// TwinCAT 3 PLC project BE_RobertWeinhandl
// ProgramVersion: 3.1.4023.0
// libraries:
//   EfficientIO Communicator, * (EfficientIO)
//   Lynus Energy Basic, * (Lynus AG)
//   Lynus Energy ModbusTCP, * (Lynus AG)
//   Lynus Standards, * (Lynus AG)
//   Tc2_MBus, * (Beckhoff Automation GmbH)
//   Tc2_Standard, * (Beckhoff Automation GmbH)
//   Tc2_System, * (Beckhoff Automation GmbH)
//   Tc2_SystemCX, * (Beckhoff Automation GmbH)
//   Tc2_Utilities, * (Beckhoff Automation GmbH)
//   Tc3_IotBase, * (Beckhoff Automation GmbH)
//   Tc3_JsonXml, * (Beckhoff Automation GmbH)
//   Tc3_Module, * (Beckhoff Automation GmbH)
// project tree:
//   / FastTask.TcTTO, MiddleTask.TcTTO, SlowTask.TcTTO
//   FB/ FB_FroniusSymo_JSON.TcPOU, FB_FroniusSymo_JSON_Helper.TcPOU, FB_KL6781_MBus_Master.TcPOU, FB_Shelly_3EM.TcPOU, FB_Shelly_3EM_Helper.TcPOU, FB_Shelly_Pro4PM.TcPOU, FB_Shelly_Pro4PM_Helper.TcPOU
//   POUs/ Logic.TcPOU (excluded from build), prgComEffIO.TcPOU, prgGrid.TcPOU, prgMain.TcPOU, prgPV.TcPOU, prgRWEffIO.TcPOU (not stored), prgShelly.TcPOU, prgSmartMeter.TcPOU (excluded from build), prgVarEffIO.TcPOU (not stored)
// real-time tasks:
//   TASK MiddleTask: cycle T#10ms, priority 8, ADS port 350
//   TASK FastTask: cycle T#5ms, priority 6, ADS port 351
//   TASK SlowTask: cycle T#20ms, priority 10, ADS port 352
// I/O:
//   DEVICE Device 1 (Beckhoff CCAT)
//   DEVICE Device 2 (CX-BK)
//     Box 1 (CX-BK)

CONFIGURATION BE_RobertWeinhandl
    RESOURCE PLC ON TwinCAT3
        TASK FastTask(INTERVAL := T#5ms, PRIORITY := 6);
        TASK MiddleTask(INTERVAL := T#10ms, PRIORITY := 8);
        TASK SlowTask(INTERVAL := T#20ms, PRIORITY := 10);
        PROGRAM prgRWEffIO WITH FastTask : prgRWEffIO;
        PROGRAM prgVarEffIO WITH FastTask : prgVarEffIO;
        PROGRAM prgShelly WITH MiddleTask : prgShelly;
        PROGRAM prgPV WITH MiddleTask : prgPV;
        PROGRAM prgGrid WITH MiddleTask : prgGrid;
        PROGRAM prgMain WITH MiddleTask : prgMain;
        PROGRAM prgComEffIO WITH SlowTask : prgComEffIO;
    END_RESOURCE
END_CONFIGURATION

// ---- POUs/prgShelly.TcPOU
PROGRAM prgShelly
VAR
	// Charging Cabel 3-phase, 400V
	fbCS						: FB_Shelly_3EM;
	
	lrPowerCSTotal				: LREAL;	//{#lynus.ag#()}
	lrPowerCSTotalkW			: LREAL;	//{#lynus.ag#()}
	lrEnergyCSTotal				: LREAL;	//{#lynus.ag#()}
	lrPowerCSL1					: LREAL;	//{#lynus.ag#()}
	lrPowerCSL2					: LREAL;	//{#lynus.ag#()}
	lrPowerCSL3					: LREAL;	//{#lynus.ag#()}
	lrCurrentCSL1				: LREAL;	//{#lynus.ag#()}
	lrCurrentCSL2				: LREAL;	//{#lynus.ag#()}
	lrCurrentCSL3				: LREAL;	//{#lynus.ag#()}
	lrVoltageCSL1				: LREAL;	//{#lynus.ag#()}
	lrVoltageCSL2				: LREAL;	//{#lynus.ag#()}
	lrVoltageCSL3				: LREAL;	//{#lynus.ag#()}
	lrEnergyCSL1				: LREAL;	//{#lynus.ag#()}
	lrEnergyCSL2				: LREAL;	//{#lynus.ag#()}
	lrEnergyCSL3				: LREAL;	//{#lynus.ag#()}
	
	// Garage and Pool
	fbGarage					: FB_Shelly_3EM;
	
	lrPowerGarageTotal			: LREAL;	//{#lynus.ag#()}
	lrPowerGarageTotalkW		: LREAL;	//{#lynus.ag#()}
	lrEnergyGarageTotal			: LREAL;	//{#lynus.ag#()}
	lrPowerGarageL1				: LREAL;	//{#lynus.ag#()}
	lrPowerGarageL2				: LREAL;	//{#lynus.ag#()}
	lrPowerGarageL3				: LREAL;	//{#lynus.ag#()}
	lrCurrentGarageL1			: LREAL;	//{#lynus.ag#()}
	lrCurrentGarageL2			: LREAL;	//{#lynus.ag#()}
	lrCurrentGarageL3			: LREAL;	//{#lynus.ag#()}
	lrVoltageGarageL1			: LREAL;	//{#lynus.ag#()}
	lrVoltageGarageL2			: LREAL;	//{#lynus.ag#()}
	lrVoltageGarageL3			: LREAL;	//{#lynus.ag#()}
	lrEnergyGarageL1			: LREAL;	//{#lynus.ag#()}
	lrEnergyGarageL2			: LREAL;	//{#lynus.ag#()}
	lrEnergyGarageL3			: LREAL;	//{#lynus.ag#()}
		
	// UV Keller
	fbUVKeller						: FB_Shelly_3EM;
	fbUVKellerCounter				: FB_EnergyCounter;
	
	lrPowerUVKellerTotal			: LREAL;	//{#lynus.ag#()}
	lrPowerUVKellerTotalkW			: LREAL;	//{#lynus.ag#()}
	lrEnergyUVKellerTotal			: LREAL;	//{#lynus.ag#()}
	lrPowerUVKellerL1				: LREAL;	//{#lynus.ag#()}
	lrPowerUVKellerL2				: LREAL;	//{#lynus.ag#()}
	lrPowerUVKellerL3				: LREAL;	//{#lynus.ag#()}
	lrCurrentUVKellerL1			: LREAL;	//{#lynus.ag#()}
	lrCurrentUVKellerL2			: LREAL;	//{#lynus.ag#()}
	lrCurrentUVKellerL3			: LREAL;	//{#lynus.ag#()}
	lrVoltageUVKellerL1			: LREAL;	//{#lynus.ag#()}
	lrVoltageUVKellerL2			: LREAL;	//{#lynus.ag#()}
	lrVoltageUVKellerL3			: LREAL;	//{#lynus.ag#()}
	lrEnergyUVKellerL1				: LREAL;	//{#lynus.ag#()}
	lrEnergyUVKellerL2				: LREAL;	//{#lynus.ag#()}
	lrEnergyUVKellerL3				: LREAL;	//{#lynus.ag#()}
END_VAR

VAR PERSISTENT
// trigger command execution
	bEnableCS 				: BOOL;		//{#lynus.ag#()}
	bEnableGarage			: BOOL;		//{#lynus.ag#()}
	bEnableUVKeller			: BOOL;		//{#lynus.ag#()}
	lrCounterUVKeller		: LREAL;	//{#lynus.ag#()}
END_VAR

// Charging Cable 3-phase, 400V
fbCS(
	bStart:= bEnableCS, 
	tDelayRequest:= T#20S, 
	sHostname:= '192.168.0.31', 
	bValidResult=> , 
	bBusy=> , 
	bError=> , 
	bDone=> , 
	hrErrorCode=> ,
	lrtotalpower=> lrPowerCSTotal,
	lrpowerL1=> lrPowerCSL1,
	lrpowerL2=> lrPowerCSL2,
	lrpowerL3=> lrPowerCSL3,
	lrcurrentL1=> lrCurrentCSL1,
	lrcurrentL2=> lrCurrentCSL2,
	lrcurrentL3=> lrCurrentCSL3,
	lrvoltageL1=> lrVoltageCSL1,
	lrvoltageL2=> lrVoltageCSL2,
	lrvoltageL3=> lrVoltageCSL3,
	lrenergyL1=> lrEnergyCSL1,
	lrenergyL2=> lrEnergyCSL2,
	lrenergyL3=> lrEnergyCSL3 );

	// re-calc to kW
	lrPowerCSTotalkW := lrPowerCSTotal / 1000;
	// sum-up energy
	lrEnergyCSTotal :=  lrEnergyCSL1 + lrEnergyCSL2 + lrEnergyCSL3;


// Garage and Pool
fbGarage(
	bStart:= bEnableGarage, 
	tDelayRequest:= T#20S, 
	sHostname:= '192.168.0.30', 
	bValidResult=> , 
	bBusy=> , 
	bError=> , 
	bDone=> , 
	hrErrorCode=> ,
	lrtotalpower=> lrPowerGarageTotal,
	lrpowerL1=> lrPowerGarageL1,
	lrpowerL2=> lrPowerGarageL2,
	lrpowerL3=> lrPowerGarageL3,
	lrcurrentL1=> lrCurrentGarageL1,
	lrcurrentL2=> lrCurrentGarageL2,
	lrcurrentL3=> lrCurrentGarageL3,
	lrvoltageL1=> lrVoltageGarageL1,
	lrvoltageL2=> lrVoltageGarageL2,
	lrvoltageL3=> lrVoltageGarageL3,
	lrenergyL1=> lrEnergyGarageL1,
	lrenergyL2=> lrEnergyGarageL2,
	lrenergyL3=> lrEnergyGarageL3 );

	// re-calc to kW
	lrPowerGarageTotalkW := lrPowerGarageTotal / 1000;
	// sum-up energy
	lrEnergyGarageTotal :=  lrEnergyGarageL1 + lrEnergyGarageL2 + lrEnergyGarageL3;

	
// UVKeller
fbUVKeller(
	bStart:= bEnableUVKeller, 
	tDelayRequest:= T#20S, 
	sHostname:= '192.168.0.35', 
	bValidResult=> , 
	bBusy=> , 
	bError=> , 
	bDone=> , 
	hrErrorCode=> ,
	lrtotalpower=> ,
	lrpowerL1=> ,
	lrpowerL2=> ,
	lrpowerL3=> ,
	lrcurrentL1=> lrCurrentUVKellerL1,
	lrcurrentL2=> lrCurrentUVKellerL2,
	lrcurrentL3=> lrCurrentUVKellerL3,
	lrvoltageL1=> lrVoltageUVKellerL1,
	lrvoltageL2=> lrVoltageUVKellerL2,
	lrvoltageL3=> lrVoltageUVKellerL3,
	lrenergyL1=> lrEnergyUVKellerL1,
	lrenergyL2=> lrEnergyUVKellerL2,
	lrenergyL3=> lrEnergyUVKellerL3 );
	
lrPowerUVKellerTotal := fbUVKeller.lrtotalpower * (-1);

	// re-calc to kW
	lrPowerUVKellerTotalkW := lrPowerUVKellerTotal / 1000;

// EnergyCounter UV Keller
fbUVKellerCounter(
	byActiveTariff:= 1, 
	lrPowerInput:= lrPowerUVKellerTotalkW, 
	lrTotalCounterEnergy_Consumption=> , 
	lrTotalCounterEnergy_Production=> , 
	lrCounterEnergyT1_Consumption=> , 
	lrCounterEnergyT2_Consumption=> , 
	lrCounterEnergyT1_Production=> , 
	lrCounterEnergyT2_Production=> );
	
IF fbUVKellerCounter.lrTotalCounterEnergy_Consumption > lrCounterUVKeller THEN  	
	lrCounterUVKeller := fbUVKellerCounter.lrTotalCounterEnergy_Consumption;
END_IF

END_PROGRAM

// ---- FB/FB_Shelly_3EM.TcPOU
FUNCTION_BLOCK FB_Shelly_3EM
VAR_INPUT
	bStart				: BOOL;
	tDelayRequest		: TIME;		//Timer for delay before start with the next read or write Request
	sHostname			: STRING(255);		//Hostname or IP Adress from the Server
END_VAR

VAR_IN_OUT
END_VAR

VAR_OUTPUT
	bValidResult		: BOOL;							//Valid Result received from Server
    bBusy				: BOOL;							//Function is Busy
    bError				: BOOL;							//Error sucess
	bDone				: BOOL;							//True after the decoding from the received Json File
	bConnected			: BOOL;							//Connection to the Server
	lrtotalpower		: LREAL;						//Received Value
	lrpowerL1			: LREAL;
	lrcurrentL1			: LREAL;
	lrvoltageL1			: LREAL;
	lrenergyL1			: LREAL;
	lrpowerL2			: LREAL;
	lrcurrentL2			: LREAL;
	lrvoltageL2			: LREAL;
	lrenergyL2			: LREAL;
	lrpowerL3			: LREAL;
	lrcurrentL3			: LREAL;
	lrvoltageL3			: LREAL;
	lrenergyL3			: LREAL;
	hrErrorCode       	: HRESULT;						//Error Result from Http Client
END_VAR

VAR
	fbClient			: FB_IotHttpClient;
	fbHttpGet			: FB_Shelly_3EM_Helper;
	timStartRequest		: TON;							//Timer to Start the Request
	FPStartRequest		: R_TRIG;						//Internal positive Edge
	FPDone				: R_TRIG;						//Internal positive Edge
	FNStart				: F_TRIG;						//Internal negative Edge
END_VAR

(*------------------------------------------------------------------------------------Configure HTTP Client------------------------------------------------------------------------------------------------------*)

fbClient.sHostName := sHostname;
fbClient.tConnectionTimeout := T#30S;

IF NOT fbClient.bConfigured THEN 
	fbClient.nHostPort:= 80;
	fbClient.bKeepAlive := TRUE;
	fbClient.tConnectionTimeout := T#30S;
END_IF


//Timer to start the Request
FPStartRequest(CLK:= bStart, Q=> );
	timStartRequest(IN:= fbClient.bConfigured AND bStart AND NOT timStartRequest.Q, PT:= tDelayRequest, Q=> , ET=> );
		IF ((timStartRequest.Q AND NOT bBusy) OR (FPStartRequest.Q AND NOT bBusy AND fbClient.bConfigured)) THEN fbHttpGet.bSend := TRUE; END_IF

				
//Http Get Function
fbHttpGet(
	lrtotalpower => lrtotalpower, 
	lrpowerL1 => lrpowerL1,
	lrcurrentL1 => lrcurrentL1,
	lrvoltageL1 => lrvoltageL1,
	lrenergyL1 => lrenergyL1,
	lrpowerL2 => lrpowerL2,
	lrcurrentL2 => lrcurrentL2,
	lrvoltageL2 => lrvoltageL2,
	lrenergyL2 => lrenergyL2,
	lrpowerL3 => lrpowerL3,
	lrcurrentL3 => lrcurrentL3,
	lrvoltageL3 => lrvoltageL3,
	lrenergyL3 => lrenergyL3,
	bSend:= , 
	fbClient:= fbClient, 
	bBusy=> bBusy, 
	bError=> ,
	sContentStatus=> ,
	sContentM0=> ,
	sContentM1=> ,
	sContentM2=> );


fbHttpGet.bSend := FALSE;

FPDone(CLK:= bDone, Q=> );

(*
//Http Client
FNStart(CLK:= bStart, Q=> );
	IF FNStart.Q THEN fbClient.Disconnect(); END_IF
*)

fbClient.Execute();

//Error
IF fbHttpGet.bError OR fbClient.bError THEN bError := TRUE; ELSE bError := FALSE; END_IF	
	hrErrorCode := fbClient.hrErrorCode;

END_FUNCTION_BLOCK

// ---- FB/FB_Shelly_3EM_Helper.TcPOU
FUNCTION_BLOCK FB_Shelly_3EM_Helper
VAR_INPUT
	bSend				: BOOL;
END_VAR

VAR_IN_OUT
	fbClient			: FB_IotHttpClient;
END_VAR

VAR_OUTPUT
	bBusy				: BOOL;
	bError				: BOOL;
	lrtotalpower		: LREAL;
	lrpowerL1			: LREAL;
	lrcurrentL1			: LREAL;
	lrvoltageL1			: LREAL;
	lrenergyL1			: LREAL;
	lrpowerL2			: LREAL;
	lrcurrentL2			: LREAL;
	lrvoltageL2			: LREAL;
	lrenergyL2			: LREAL;
	lrpowerL3			: LREAL;
	lrcurrentL3			: LREAL;
	lrvoltageL3			: LREAL;
	lrenergyL3			: LREAL;
END_VAR

VAR
	fbRequestStatus		: FB_IotHttpRequest;
	fbRequestMeter0		: FB_IotHttpRequest;
	fbRequestMeter1		: FB_IotHttpRequest;
	fbRequestMeter2		: FB_IotHttpRequest;
	fbJson				: FB_JsonDomParser;
	nState				: UDINT;
	RisingEdge			: R_TRIG;
	timTimeout			: TON;
	tTimeOut			: TIME := T#50S;
	bGetContentResult	: BOOL;
	sContentStatus		: STRING(511);
	sContentM0			: STRING(511);
	sContentM1			: STRING(511);
	sContentM2			: STRING(511);
	
	bGetJsonResult		: BOOL;
	jsonDoc				: SJsonValue;
	jsonVal				: SJsonValue;
	
	nReqCount			: UDINT;	
	nResCount			: UDINT;
	nValidResCount		: UDINT;
	nErrCount			: UDINT;
END_VAR

//Timer for Timeout
timTimeout(IN:= nState = 1 AND bBusy, PT:= tTimeOut, Q=> , ET=> );
	IF timTimeout.Q THEN 
		nState := 0;
		bBusy := FALSE;
	END_IF

RisingEdge(CLK:= bSend );
CASE nState OF
0:	
	IF RisingEdge.Q THEN 
		IF 
			fbRequestStatus.SendRequest(sUri:='/status', fbClient:=fbClient, eRequestType:=ETcIotHttpRequestType.HTTP_Get, 0, 0, 0) AND
			fbRequestMeter0.SendRequest(sUri:='/emeter/0', fbClient:=fbClient, eRequestType:=ETcIotHttpRequestType.HTTP_Get, 0, 0, 0) AND 
			fbRequestMeter1.SendRequest(sUri:='/emeter/1', fbClient:=fbClient, eRequestType:=ETcIotHttpRequestType.HTTP_Get, 0, 0, 0) AND
			fbRequestMeter2.SendRequest(sUri:='/emeter/2', fbClient:=fbClient, eRequestType:=ETcIotHttpRequestType.HTTP_Get, 0, 0, 0) THEN				
			nState:= 1;
			nReqCount:= nReqCount+1;
			bBusy:= TRUE;
			bError:= FALSE;
		END_IF					
	END_IF
1:
	IF NOT fbRequestMeter0.bBusy AND NOT fbRequestMeter1.bBusy AND NOT fbRequestMeter2.bBusy AND NOT fbRequestStatus.bBusy THEN
		bError:= TRUE;
		IF NOT fbRequestMeter0.bError THEN				 
			bGetContentResult:= fbRequestMeter0.GetContent(pContent:= ADR(sContentM0), nContentSize:= SIZEOF(sContentM0), bSetNullTermination:= TRUE);
			IF fbRequestMeter0.nStatusCode >= 200 AND fbRequestMeter0.nStatusCode < 300 THEN
				bGetJsonResult:= FALSE;
				jsonDoc:= fbRequestMeter0.GetJsonDomContent(fbJson);
				IF jsonDoc <> 0 THEN
					bGetJsonResult:= TRUE;
					IF fbJson.HasMember(jsonDoc, 'power')  THEN
						jsonVal:= fbJson.FindMember(jsonDoc, 'power');
						nValidResCount:= nValidResCount+1;
						IF fbJson.IsDouble(jsonVal) THEN							
							lrpowerL1:= fbJson.GetDouble(jsonVal);									
						END_IF
						jsonVal:= fbJson.FindMember(jsonDoc, 'current');
						nValidResCount:= nValidResCount+1;
						IF fbJson.IsDouble(jsonVal) THEN							
							lrcurrentL1:= fbJson.GetDouble(jsonVal);									
						END_IF
						jsonVal:= fbJson.FindMember(jsonDoc, 'voltage');
						nValidResCount:= nValidResCount+1;
						IF fbJson.IsDouble(jsonVal) THEN							
							lrvoltageL1:= fbJson.GetDouble(jsonVal);									
						END_IF
						jsonVal:= fbJson.FindMember(jsonDoc, 'total');
						nValidResCount:= nValidResCount+1;
						IF fbJson.IsDouble(jsonVal) THEN							
							lrenergyL1:= fbJson.GetDouble(jsonVal);									
						END_IF	
						bError:= FALSE;
						END_IF
					END_IF						
				nResCount:= nResCount+1;			
				END_IF
		END_IF
		
		IF NOT fbRequestMeter1.bError THEN				 
			bGetContentResult:= fbRequestMeter1.GetContent(pContent:= ADR(sContentM1), nContentSize:= SIZEOF(sContentM1), bSetNullTermination:= TRUE);
			IF fbRequestMeter1.nStatusCode >= 200 AND fbRequestMeter1.nStatusCode < 300 THEN
				bGetJsonResult:= FALSE;
				jsonDoc:= fbRequestMeter1.GetJsonDomContent(fbJson);
				IF jsonDoc <> 0 THEN
					bGetJsonResult:= TRUE;
					IF fbJson.HasMember(jsonDoc, 'power')  THEN
						jsonVal:= fbJson.FindMember(jsonDoc, 'power');
						nValidResCount:= nValidResCount+1;
						IF fbJson.IsDouble(jsonVal) THEN							
							lrpowerL2:= fbJson.GetDouble(jsonVal);									
						END_IF
						jsonVal:= fbJson.FindMember(jsonDoc, 'current');
						nValidResCount:= nValidResCount+1;
						IF fbJson.IsDouble(jsonVal) THEN							
							lrcurrentL2:= fbJson.GetDouble(jsonVal);									
						END_IF
						jsonVal:= fbJson.FindMember(jsonDoc, 'voltage');
						nValidResCount:= nValidResCount+1;
						IF fbJson.IsDouble(jsonVal) THEN							
							lrvoltageL2:= fbJson.GetDouble(jsonVal);									
						END_IF
						jsonVal:= fbJson.FindMember(jsonDoc, 'total');
						nValidResCount:= nValidResCount+1;
						IF fbJson.IsDouble(jsonVal) THEN							
							lrenergyL2:= fbJson.GetDouble(jsonVal);									
						END_IF	
						bError:= FALSE;
						END_IF
					END_IF						
				nResCount:= nResCount+1;			
				END_IF
		END_IF
		
		IF NOT fbRequestMeter2.bError THEN				 
			bGetContentResult:= fbRequestMeter2.GetContent(pContent:= ADR(sContentM2), nContentSize:= SIZEOF(sContentM2), bSetNullTermination:= TRUE);
			IF fbRequestMeter2.nStatusCode >= 200 AND fbRequestMeter2.nStatusCode < 300 THEN
				bGetJsonResult:= FALSE;
				jsonDoc:= fbRequestMeter2.GetJsonDomContent(fbJson);
				IF jsonDoc <> 0 THEN
					bGetJsonResult:= TRUE;
					IF fbJson.HasMember(jsonDoc, 'power')  THEN
						jsonVal:= fbJson.FindMember(jsonDoc, 'power');
						nValidResCount:= nValidResCount+1;
						IF fbJson.IsDouble(jsonVal) THEN							
							lrpowerL3:= fbJson.GetDouble(jsonVal);									
						END_IF
						jsonVal:= fbJson.FindMember(jsonDoc, 'current');
						nValidResCount:= nValidResCount+1;
						IF fbJson.IsDouble(jsonVal) THEN							
							lrcurrentL3:= fbJson.GetDouble(jsonVal);									
						END_IF
						jsonVal:= fbJson.FindMember(jsonDoc, 'voltage');
						nValidResCount:= nValidResCount+1;
						IF fbJson.IsDouble(jsonVal) THEN							
							lrvoltageL3:= fbJson.GetDouble(jsonVal);									
						END_IF
						jsonVal:= fbJson.FindMember(jsonDoc, 'total');
						nValidResCount:= nValidResCount+1;
						IF fbJson.IsDouble(jsonVal) THEN							
							lrenergyL3:= fbJson.GetDouble(jsonVal);									
						END_IF	
						bError:= FALSE;
						END_IF
					END_IF						
				nResCount:= nResCount+1;			
				END_IF
		END_IF
		
		IF NOT fbRequestStatus.bError THEN				 
			bGetContentResult:= fbRequestStatus.GetContent(pContent:= ADR(sContentStatus), nContentSize:= SIZEOF(sContentStatus), bSetNullTermination:= TRUE);
			IF fbRequestStatus.nStatusCode >= 200 AND fbRequestStatus.nStatusCode < 300 THEN
				bGetJsonResult:= FALSE;
				jsonDoc:= fbRequestStatus.GetJsonDomContent(fbJson);
				IF jsonDoc <> 0 THEN
					bGetJsonResult:= TRUE;
					IF fbJson.HasMember(jsonDoc, 'total_power')  THEN
						jsonVal:= fbJson.FindMember(jsonDoc, 'total_power');
						nValidResCount:= nValidResCount+1;
						IF fbJson.IsDouble(jsonVal) THEN							
							lrtotalpower:= fbJson.GetDouble(jsonVal);									
						END_IF
						bError:= FALSE;
					END_IF
				END_IF		
				nResCount:= nResCount+1;			
			END_IF
		END_IF
		
		nState:= 0;
		bBusy:= FALSE;
		IF bError THEN
			nErrCount:= nErrCount+1;
		END_IF
	END_IF  	
END_CASE

END_FUNCTION_BLOCK

// ---- POUs/prgPV.TcPOU
PROGRAM prgPV
VAR
	fbPV					: FB_Symo_PV_Inverter_FLOAT_1_DM_1_Inverter;
	fbPVInt					: FB_PV_Power;
	fbPVCounter				: FB_EnergyCounter;
	lrPowerPV				: LREAL;				//{#lynus.ag#()}
	byErrorWarningPV		: BYTE;					//{#lynus.ag#()}
	bReadyPD_PV				: BOOL;					//{#lynus.ag#()}
	byErrorWarningPD_PV		: BYTE;					//{#lynus.ag#()}
	rHeartbeat_PD_PV		: REAL;					//{#lynus.ag#()}
END_VAR

VAR PERSISTENT
	lrCounterPV				: LREAL;				//{#lynus.ag#()}
END_VAR

fbPV(
	bEnable:= TRUE, 
	sIPAdress:= '192.168.0.102', 
	byUnitID_Inverter:= 1, 
	stDataSymo10=> , 
	stDataEMPower_PV=> , 
	stDataEMCounter_PV=> , 
	diNrOfEM_OUT_PV=> );

fbPVInt(
	bEnable:= TRUE, 
	bPowerDataInvers:= , 
	diNrOfEM_IN_PV:= fbPV.diNrOfEM_OUT_PV, 
	stDataPv=> , 
	diNrOfPv_OUT=> );
	
lrPowerPV := fbPVInt.stDataPv.lrPower;
	byErrorWarningPV := fbPVInt.stDataPv.byErrorWarning;

// EnergyCounter
fbPVCounter(
	byActiveTariff:= 1, 
	lrPowerInput:= 0 - lrPowerPV, 
	lrTotalCounterEnergy_Consumption=> , 
	lrTotalCounterEnergy_Production=> , 
	lrCounterEnergyT1_Consumption=> , 
	lrCounterEnergyT2_Consumption=> , 
	lrCounterEnergyT1_Production=> , 
	lrCounterEnergyT2_Production=> );
	
IF fbPVCounter.lrTotalCounterEnergy_Production > lrCounterPV THEN  	
	lrCounterPV := fbPVCounter.lrTotalCounterEnergy_Production;
END_IF

END_PROGRAM

// ---- POUs/prgGrid.TcPOU
PROGRAM prgGrid
VAR
	lrPowerGridkW		: LREAL;	//{#lynus.ag#()}
END_VAR

lrPowerGridkW := prgShelly.lrPowerCSTotalkW + prgShelly.lrPowerGarageTotalkW + prgShelly.lrPowerUVKellerTotalkW - prgPV.lrPowerPV;

END_PROGRAM

// ---- POUs/prgMain.TcPOU
PROGRAM prgMain
VAR
	fb_Reboot		: NT_reboot;
	m_Reboot		: BOOL:=FALSE;
END_VAR

fb_Reboot(	netid := '',
			delay := 2,
			start := m_Reboot);

END_PROGRAM

// ---- POUs/prgComEffIO.TcPOU
PROGRAM prgComEffIO
VAR
	fbCom		: FB_MqttCommunicator_V2;
END_VAR

fbCom(
	bConnect:= TRUE, 
	strAuthKey := 'BE736352867778',
	sUserName:= '9e35a788-9544-4d1e-a992-8e2eed9a2bf4', 
	sUserPassword:= 'b22fd0d3-05b2-481b-ab97-9bb6cc09e5f2', 
	eSavePositionCertificate:= eSavePositionOnPLC.ePostionHardDisk, 
	bConnected=> , 
	bError=> , 
	hrErrorCode=> , 
	eConnectionState=> , 
	eErrorMessage_Out=> );

END_PROGRAM

// ---- FB/FB_FroniusSymo_JSON.TcPOU
FUNCTION_BLOCK FB_FroniusSymo_JSON
VAR_INPUT
	bStart				: BOOL;
	tDelayRequest		: TIME := T#3S;	//Timer for delay before start with the next read or write Request
	sHostname			: STRING(255);		//Hostname or IP Adress from the Server
END_VAR

VAR_IN_OUT
END_VAR

VAR_OUTPUT
	bValidResult				: BOOL;															//Valid Result received from Server
    bBusy						: BOOL;															//Function is Busy
    bError						: BOOL;															//Error sucess
	bDone						: BOOL;															//True after the decoding from the received Json File
	bConnected					: BOOL;															//Connection to the Server
	lrpowerP1					: LREAL;														//Received Value
	lrvoltageP1					: LREAL;														//Received Value
	lrenergyP1					: LREAL;														//Received Value
	lrpowerP2					: LREAL;														//Received Value
	lrvoltageP2					: LREAL;														//Received Value
	lrenergyP2					: LREAL;
	lrpowerP3					: LREAL;														//Received Value
	lrvoltageP3					: LREAL;														//Received Value
	lrenergyP3					: LREAL;
	lrpowerP4					: LREAL;														//Received Value
	lrvoltageP4					: LREAL;														//Received Value
	lrenergyP4					: LREAL;	
	hrErrorCode       			: HRESULT;														//Error Result from Http Client
END_VAR

VAR
	fbClient					: FB_IotHttpClient;
	fbHttpGet					: FB_FroniusSymo_JSON_Helper;
	timStartRequest				: TON;															//Timer to Start the Request
	FPStartRequest				: R_TRIG;														//Internal positive Edge
	FPDone						: R_TRIG;														//Internal positive Edge
	FNStart						: F_TRIG;														//Internal negative Edge
END_VAR

(*------------------------------------------------------------------------------------Configure HTTP Client------------------------------------------------------------------------------------------------------*)

fbClient.sHostName := sHostname;
fbClient.tConnectionTimeout := tDelayRequest;

IF NOT fbClient.bConfigured THEN 
	fbClient.nHostPort:= 80;
	fbClient.bKeepAlive := TRUE;
	fbClient.tConnectionTimeout := T#2S;
END_IF


//Timer to start the Request
FPStartRequest(CLK:= bStart, Q=> );
	timStartRequest(IN:= fbClient.bConfigured AND bStart AND NOT timStartRequest.Q, PT:= tDelayRequest, Q=> , ET=> );
		IF ((timStartRequest.Q AND NOT bBusy) OR (FPStartRequest.Q AND NOT bBusy AND fbClient.bConfigured)) THEN fbHttpGet.bSend := TRUE; END_IF

				
//Http Get Function
fbHttpGet(
	lrapowerP1 => lrpowerP1, 
	lrvoltageP1 => lrvoltageP1, 
	lraenergyP1 => lrenergyP1,
	lrapowerP2 => lrpowerP2, 
	lrvoltageP2 => lrvoltageP2, 
	lraenergyP2 => lrenergyP2,
	lrapowerP3 => lrpowerP3, 
	lrvoltageP3 => lrvoltageP3, 
	lraenergyP3 => lrenergyP3,
	lrapowerP4 => lrpowerP4, 
	lrvoltageP4 => lrvoltageP4, 
	lraenergyP4 => lrenergyP4, 
	bSend:= , 
	fbClient:= fbClient, 
	bBusy=> bBusy, 
	bError=> ,
	sContentS0=> ,
	sContentS1=> ,
	sContentS2=> ,
	sContentS3=> );


fbHttpGet.bSend := FALSE;

FPDone(CLK:= bDone, Q=> );

//Http Client
FNStart(CLK:= bStart, Q=> );
	IF FNStart.Q THEN fbClient.Disconnect(); END_IF

fbClient.Execute();

//Error
IF fbHttpGet.bError OR fbClient.bError THEN bError := TRUE; ELSE bError := FALSE; END_IF	
	hrErrorCode := fbClient.hrErrorCode;

END_FUNCTION_BLOCK

// ---- FB/FB_FroniusSymo_JSON_Helper.TcPOU
FUNCTION_BLOCK FB_FroniusSymo_JSON_Helper
VAR_INPUT
	bSend			: BOOL;
END_VAR

VAR_IN_OUT
	fbClient		: FB_IotHttpClient;
END_VAR

VAR_OUTPUT
	bBusy			: BOOL;
	bError			: BOOL;
	lrapowerP1		: LREAL;
	lrvoltageP1		: LREAL;
	lraenergyP1		: LREAL;
	lrapowerP2		: LREAL;
	lrvoltageP2		: LREAL;
	lraenergyP2		: LREAL;
	lrapowerP3		: LREAL;
	lrvoltageP3		: LREAL;
	lraenergyP3		: LREAL;
	lrapowerP4		: LREAL;
	lrvoltageP4		: LREAL;
	lraenergyP4		: LREAL;
END_VAR

VAR
	fbRequestSwitch0	: FB_IotHttpRequest;
	fbRequestSwitch1	: FB_IotHttpRequest;
	fbRequestSwitch2	: FB_IotHttpRequest;
	fbRequestSwitch3	: FB_IotHttpRequest;
	fbJson				: FB_JsonDomParser;
	fbPayload			: FB_JsonSaxWriter;
	fbHeader            : FB_IotHttpHeaderFieldMap;
	nState				: UDINT;
	RisingEdge			: R_TRIG;
	
	bGetContentResult	: BOOL;
	bOnce				: BOOL;
	sContent			: STRING(511);
	sContentS0			: STRING(2048);
	sContentS1			: STRING(511);
	sContentS2			: STRING(511);
	sContentS3			: STRING(511);
	
	bGetJsonResult		: BOOL;
	jsonDoc				: SJsonValue;
	jsonVal				: SJsonValue;
	
	nReqCount			: UDINT;	
	nResCount			: UDINT;
	nValidResCount		: UDINT;
	nErrCount			: UDINT;
END_VAR

IF bOnce THEN
	fbHeader.AddField('Content-type','application/json', FALSE);
	bOnce:= FALSE;
END_IF

RisingEdge(CLK:= bSend );
CASE nState OF
0:	
	IF RisingEdge.Q THEN 
		IF
			fbRequestSwitch0.SendRequest(sUri:='/solar_api/v1/GetInverterRealtimeData.cgi?Scope=Device&DeviceID=1&DataCollection=CommonInverterData', fbClient:=fbClient, eRequestType:=ETcIotHttpRequestType.HTTP_Get, 0, 0, fbHeader) THEN				
			nState:= 1;
			nReqCount:= nReqCount+1;
			bBusy:= TRUE;
			bError:= FALSE;
		END_IF					
	END_IF
1:
	IF NOT fbRequestSwitch0.bBusy THEN
		bError:= TRUE;
		
		IF NOT fbRequestSwitch0.bError THEN				 
			bGetContentResult:= fbRequestSwitch0.GetContent(pContent:= ADR(sContentS0), nContentSize:= SIZEOF(sContentS0), bSetNullTermination:= TRUE);
			IF fbRequestSwitch0.nStatusCode >= 200 AND fbRequestSwitch0.nStatusCode < 300 THEN
				bGetJsonResult:= FALSE;
				//sResponseContent := 
				jsonDoc:= fbRequestSwitch0.GetJsonDomContent(fbJson);
				IF jsonDoc <> 0 THEN
					bGetJsonResult:= TRUE;
					IF fbJson.HasMember(jsonDoc, 'Body')  THEN
						jsonVal:= fbJson.FindMember(jsonDoc, 'Body');
                        IF fbJson.HasMember(jsonVal, 'Data') THEN
                            jsonVal:= fbJson.FindMember(jsonVal, 'Data');
								IF fbJson.HasMember(jsonVal, 'PAC') THEN
									jsonVal:= fbJson.FindMember(jsonVal, 'PAC');
										IF fbJson.HasMember(jsonVal, 'Value') THEN
											jsonVal:= fbJson.FindMember(jsonVal, 'Value');
										END_IF
								END_IF	
						END_IF
					END_IF
				END_IF
			nValidResCount:= nValidResCount+1;
			IF fbJson.IsDouble(jsonVal) THEN
				lraenergyP1:= fbJson.GetDouble(jsonVal);
			END_IF
			bError:= FALSE;
			nResCount:= nResCount+1;
			END_IF
		END_IF						
					
	nState:= 0;
	bBusy:= FALSE;
		IF bError THEN
			nErrCount:= nErrCount+1;
		END_IF
	END_IF  	
END_CASE

fbClient.Execute();

END_FUNCTION_BLOCK

// ---- FB/FB_KL6781_MBus_Master.TcPOU
FUNCTION_BLOCK FB_KL6781_MBus_Master
VAR_INPUT PERSISTENT
	eBaudrateMBus							: E_MBus_Baudrate;				//With this Baudrate the Functionsblocks for the Counters are reading out
END_VAR
VAR_OUTPUT
	bBusy									: BOOL;							//Function is Busy
	bReady									: BOOL;							//Function is Ready
	byErrorWarning							: BYTE;							//Error Warning State
	diNrOfMBusMasterLine_OUT				: DINT;							//Active Number from the MBus Master Function for using on other functions
	eMessageMBusMaster						: E_Message_MBusMaster;			//Message from the MBus Master Function
END_VAR
VAR

	fbMbusMaster							: FB_MBUSKL6781;				//MBus Master for KL6781
	fbNumberDevice							: FB_NumberOfDevice;			//Function block to calcualte the number of the Device
	fbMBusMessage							: FB_MBusMaster_Messages;		//MBus Messages
	fbPD									: FB_PersistentData_Number;		//FB Persistent Data
	timDissableFunctions					: TON;							//Timer to dissable the Function after Lynus_Standards.Constants_General.tTimeDissableLynusFunctions Days without connection to the Lynus Cloud
	timResetConnectionOnGVL					: TON;							//Timer to try reset the connection Flag on the GVL. (When somebody delete the Connection Function and make only a onlinechange)
	stMBusKL6781ComIn        	AT%I*	 	: ST_KL6781inData22B;			//Input Structure for the KL6781 to map on the KL6781 Terminal
	stMBusKL6781ComOut        	AT%Q*		: ST_KL6781outData22B;			//Output Structure for the KL6781 to map on the KL6781 Terminal
	byWaitInStep							: BYTE;							//Wait in Step before start to clean data on PLC
	iStateGVLData							: INT;							//State machine to handle the data on the GVL
	diCounterForGVL							: DINT;							//Counter to clean old data on GVL
END_VAR

//Creator : Kai Ebensperger
//Company : Lynus AG
//Date : 23.07.2021
//Version : 1.0.0.0

//With this function block we can communicate with a beckhoff KL6781 MBus Terminal.
//This Functionblock receive the requests from the other Counter Functions and send to the Hardware Counters in the field.
//The answer from the Hardware Counters comes back to this Function and then they distribute to the Counter Function in the plc.
//This Function must be called in a task of < 10MS. Is depends about the Baudrate. 2400Baud = 10MS Task
//The request to a Hardware counter and the response is min. 1 second on MBus.


//NOTE for diNr.....Designation => 
//_IN = Here Data come in from other Functions or go out to other functions about the GVL
//_OUT = Here Data go out to other functions about the GVL

(*-------------------------------------------------------------Calcualte the number of MBus Master---------------------------------------------------------------*)

fbNumberDevice(
	diActualNumberOfDevices:= Lynus_Standards.GVL_Bussystems.diNumberOfMBusMasters, 
	diMaxNumberOfDevices:= Constants_Bussystems.diMaxNumberOfMBusMasterKL6781, 
	udiCounterOnlineChange:= TwinCAT_SystemInfoVarList._AppInfo.OnlineChangeCnt, 
	bNumberIsCalculatet=> , 
	bFPNumberIsCalculatet=> , 
	bOnlineChange=> , 
	diNumberForThisDevice=> diNrOfMBusMasterLine_OUT, 
	diNumberOfTotalDevices=> );

//Write new Numer on GVL
IF fbNumberDevice.bFPNumberIsCalculatet THEN
	Lynus_Standards.GVL_Bussystems.diNumberOfMBusMasters := fbNumberDevice.diNumberOfTotalDevices;	
END_IF 

//Delete old Number on GVL
IF fbNumberDevice.bOnlineChange THEN 
	Lynus_Standards.GVL_Bussystems.diNumberOfMBusMasters := diNrOfMBusMasterLine_OUT;	
		iStateGVLData := 1; 
END_IF	

(*-------------------------------------------------------------Service from Backend is ready and check the connection to backen for dissabel/enable Function---------------------------------------------------------------*)

//Try to reset the variable for connection on the GVL. When all is normal then the Lynus Mqtt connection function set this variable to true in the next cycle
//When we have no connection to the backend then after Lynus_Standards.Constants_General.tTimeDissableLynusFunctions days the Function is dissabled with all of his functionalities
timResetConnectionOnGVL(IN:= NOT timResetConnectionOnGVL.Q, PT:= T#1H, Q=> , ET=> );
	IF timResetConnectionOnGVL.Q THEN Lynus_Standards.GVL_Communicator.bStateConnectionToEnableFunctions := FALSE; END_IF
		IF NOT Lynus_Standards.GVL_Communicator.bStateConnectionToEnableFunctions THEN timDissableFunctions.IN := TRUE; ELSE timDissableFunctions.IN := FALSE; END_IF  
			timDissableFunctions(IN:= , PT:= Lynus_Standards.Constants_General.tTimeDissableLynusFunctions, Q=> , ET=> );
			
(*-------------------------------------------------------------M-Bus Master---------------------------------------------------------------*)

fbMbusMaster(
	usiRetries:= 0, 
	bStart:= , 
	bDisabled:= timDissableFunctions.Q OR diNrOfMBusMasterLine_OUT <= 0 OR NOT fbNumberDevice.bNumberIsCalculatet , 
	bBusy=> bBusy, 
	bReady=> bReady, 
	bError=> , 
	eError=> , 
	stComIn:= stMBusKL6781ComIn, 
	stComOut:= stMBusKL6781ComOut, 
	stCom:= Lynus_Standards.GVL_Bussystems.stDataOfMBusMasterKL6781[diNrOfMBusMasterLine_OUT].stDataMBusCommunicationKL6781);
	
(*------------------------------------------------------------------Error and Warning----------------------------------------------------------------------------*)
			
IF timDissableFunctions.Q THEN fbMBusMessage.bWarning := TRUE; fbMBusMessage.iWarningCode := 0; ELSE fbMBusMessage.bWarning := FALSE; END_IF   
	IF (Lynus_Standards.GVL_Bussystems.diNumberOfMBusMasters > Constants_Bussystems.diMaxNumberOfMBusMasterKL6781) THEN 
		fbMBusMessage.bErrorIntern := TRUE;
			fbMBusMessage.iErrorCode := 1;
	ELSE
		fbMBusMessage.bErrorIntern := FALSE;
	END_IF	

IF fbMbusMaster.bError THEN 
	fbMBusMessage.bErrorMBus := TRUE;
		fbMBusMessage.iErrorCode := fbMbusMaster.eError;
ELSE
	IF NOT fbMbusMaster.bError AND NOT fbMbusMaster.bBusy THEN 
		fbMBusMessage.bErrorMBus := FALSE;
	END_IF
END_IF	
		
fbMBusMessage(
	bErrorMBus:= , 
	bErrorIntern:= , 
	bWarning:= , 
	iWarningCode:= , 
	iErrorCode:= , 
	byErrorWarning=> byErrorWarning, 
	eMessageMBusMaster=> eMessageMBusMaster);
	
(*-----------------------------------------------------------Handle data to Global structure for MBus Communication-----------------------------------------------------------------*)
	
CASE iStateGVLData OF
	
	0://Init Step
		byWaitInStep := 0;
			diCounterForGVL := 1;
	
	1://Wait for 4 Steps before clean al Data on GVL
		byWaitInStep := byWaitInStep + 1;
			IF byWaitInStep >= 4 AND fbNumberDevice.bNumberIsCalculatet THEN iStateGVLData := 2; END_IF
				//To much Devices, back to the Init step
				IF byWaitInStep >= 4 AND NOT fbNumberDevice.bNumberIsCalculatet THEN iStateGVLData := 0; END_IF	
			
	2://Clear all Data in GVL
	//Some Parts in the GVL Reset the Slave. Otherwise there will be problems when writing the new addresses to the array in the GVL.
	
		Lynus_Standards.GVL_Bussystems.stDataOfMBusMasterKL6781[diCounterForGVL].eBaudrateMBusKL6781 := E_MBus_Baudrate.eMBus_NoBaudrate;
														 		
		diCounterForGVL := diCounterForGVL + 1;
			diCounterForGVL := LIMIT(0,diCounterForGVL,Constants_Bussystems.diMaxNumberOfMBusMasterKL6781);
				//Back to the init step
				IF diCounterForGVL >= Constants_Bussystems.diMaxNumberOfMBusMasterKL6781 THEN iStateGVLData := 0; END_IF

END_CASE 
	
IF diNrOfMBusMasterLine_OUT > 0 AND fbNumberDevice.bNumberIsCalculatet THEN  
	Lynus_Standards.GVL_Bussystems.stDataOfMBusMasterKL6781[diNrOfMBusMasterLine_OUT].eBaudrateMBusKL6781 := eBaudrateMBus;
END_IF	

(*----------------------------------------------------------Save persistent data----------------------------------------------------------------*)

fbPD(lrValue:= INT_TO_LREAL(eBaudrateMBus), bEventBasedActive=> );

END_FUNCTION_BLOCK

// ---- FB/FB_Shelly_Pro4PM.TcPOU
FUNCTION_BLOCK FB_Shelly_Pro4PM
VAR_INPUT
	bStart				: BOOL;
	tDelayRequest		: TIME := T#3S;	//Timer for delay before start with the next read or write Request
	sHostname			: STRING(255);		//Hostname or IP Adress from the Server
END_VAR

VAR_IN_OUT
END_VAR

VAR_OUTPUT
	bValidResult				: BOOL;															//Valid Result received from Server
    bBusy						: BOOL;															//Function is Busy
    bError						: BOOL;															//Error sucess
	bDone						: BOOL;															//True after the decoding from the received Json File
	bConnected					: BOOL;															//Connection to the Server
	lrpowerP1					: LREAL;														//Received Value
	lrvoltageP1					: LREAL;														//Received Value
	lrenergyP1					: LREAL;														//Received Value
	lrpowerP2					: LREAL;														//Received Value
	lrvoltageP2					: LREAL;														//Received Value
	lrenergyP2					: LREAL;
	lrpowerP3					: LREAL;														//Received Value
	lrvoltageP3					: LREAL;														//Received Value
	lrenergyP3					: LREAL;
	lrpowerP4					: LREAL;														//Received Value
	lrvoltageP4					: LREAL;														//Received Value
	lrenergyP4					: LREAL;	
	hrErrorCode       			: HRESULT;														//Error Result from Http Client
END_VAR

VAR
	fbClient					: FB_IotHttpClient;
	fbHttpGet					: FB_Shelly_Pro4PM_Helper;
	timStartRequest				: TON;															//Timer to Start the Request
	FPStartRequest				: R_TRIG;														//Internal positive Edge
	FPDone						: R_TRIG;														//Internal positive Edge
	FNStart						: F_TRIG;														//Internal negative Edge
END_VAR

(*------------------------------------------------------------------------------------Configure HTTP Client------------------------------------------------------------------------------------------------------*)

fbClient.sHostName := sHostname;
fbClient.tConnectionTimeout := tDelayRequest;

IF NOT fbClient.bConfigured THEN 
	fbClient.nHostPort:= 80;
	fbClient.bKeepAlive := TRUE;
	fbClient.tConnectionTimeout := T#2S;
END_IF


//Timer to start the Request
FPStartRequest(CLK:= bStart, Q=> );
	timStartRequest(IN:= fbClient.bConfigured AND bStart AND NOT timStartRequest.Q, PT:= tDelayRequest, Q=> , ET=> );
		IF ((timStartRequest.Q AND NOT bBusy) OR (FPStartRequest.Q AND NOT bBusy AND fbClient.bConfigured)) THEN fbHttpGet.bSend := TRUE; END_IF

				
//Http Get Function
fbHttpGet(
	lrapowerP1 => lrpowerP1, 
	lrvoltageP1 => lrvoltageP1, 
	lraenergyP1 => lrenergyP1,
	lrapowerP2 => lrpowerP2, 
	lrvoltageP2 => lrvoltageP2, 
	lraenergyP2 => lrenergyP2,
	lrapowerP3 => lrpowerP3, 
	lrvoltageP3 => lrvoltageP3, 
	lraenergyP3 => lrenergyP3,
	lrapowerP4 => lrpowerP4, 
	lrvoltageP4 => lrvoltageP4, 
	lraenergyP4 => lrenergyP4, 
	bSend:= , 
	fbClient:= fbClient, 
	bBusy=> bBusy, 
	bError=> ,
	sContentS0=> ,
	sContentS1=> ,
	sContentS2=> ,
	sContentS3=> );


fbHttpGet.bSend := FALSE;

FPDone(CLK:= bDone, Q=> );

(*
//Http Client
FNStart(CLK:= bStart, Q=> );
	IF FNStart.Q THEN fbClient.Disconnect(); END_IF
*)

fbClient.Execute();

//Error
IF fbHttpGet.bError OR fbClient.bError THEN bError := TRUE; ELSE bError := FALSE; END_IF	
	hrErrorCode := fbClient.hrErrorCode;

END_FUNCTION_BLOCK

// ---- FB/FB_Shelly_Pro4PM_Helper.TcPOU
FUNCTION_BLOCK FB_Shelly_Pro4PM_Helper
VAR_INPUT
	bSend			: BOOL;
END_VAR

VAR_IN_OUT
	fbClient		: FB_IotHttpClient;
END_VAR

VAR_OUTPUT
	bBusy			: BOOL;
	bError			: BOOL;
	lrapowerP1		: LREAL;
	lrvoltageP1		: LREAL;
	lraenergyP1		: LREAL;
	lrapowerP2		: LREAL;
	lrvoltageP2		: LREAL;
	lraenergyP2		: LREAL;
	lrapowerP3		: LREAL;
	lrvoltageP3		: LREAL;
	lraenergyP3		: LREAL;
	lrapowerP4		: LREAL;
	lrvoltageP4		: LREAL;
	lraenergyP4		: LREAL;
END_VAR

VAR
	fbRequestSwitch0	: FB_IotHttpRequest;
	fbRequestSwitch1	: FB_IotHttpRequest;
	fbRequestSwitch2	: FB_IotHttpRequest;
	fbRequestSwitch3	: FB_IotHttpRequest;
	fbJson				: FB_JsonDomParser;
	nState				: UDINT;
	RisingEdge			: R_TRIG;
	timTimeout			: TON;
	tTimeOut			: TIME := T#30S;
	
	bGetContentResult	: BOOL;
	sContentS0			: STRING(511);
	sContentS1			: STRING(511);
	sContentS2			: STRING(511);
	sContentS3			: STRING(511);
	
	bGetJsonResult		: BOOL;
	jsonDoc				: SJsonValue;
	jsonVal				: SJsonValue;
	
	nReqCount			: UDINT;	
	nResCount			: UDINT;
	nValidResCount		: UDINT;
	nErrCount			: UDINT;
END_VAR

//Timer for Timeout
timTimeout(IN:= nState = 1 AND bBusy, PT:= tTimeOut, Q=> , ET=> );
	IF timTimeout.Q THEN 
		nState := 0;
		bBusy := FALSE;
	END_IF

RisingEdge(CLK:= bSend );
CASE nState OF
0:	
	IF RisingEdge.Q THEN 
		IF
			fbRequestSwitch0.SendRequest(sUri:='/rpc/Switch.GetStatus?id=0', fbClient:=fbClient, eRequestType:=ETcIotHttpRequestType.HTTP_Get, 0, 0, 0) AND
			fbRequestSwitch1.SendRequest(sUri:='/rpc/Switch.GetStatus?id=1', fbClient:=fbClient, eRequestType:=ETcIotHttpRequestType.HTTP_Get, 0, 0, 0) AND
			fbRequestSwitch2.SendRequest(sUri:='/rpc/Switch.GetStatus?id=2', fbClient:=fbClient, eRequestType:=ETcIotHttpRequestType.HTTP_Get, 0, 0, 0) AND
			fbRequestSwitch3.SendRequest(sUri:='/rpc/Switch.GetStatus?id=3', fbClient:=fbClient, eRequestType:=ETcIotHttpRequestType.HTTP_Get, 0, 0, 0) THEN				
			nState:= 1;
			nReqCount:= nReqCount+1;
			bBusy:= TRUE;
			bError:= FALSE;
		END_IF					
	END_IF
1:
	IF NOT fbRequestSwitch0.bBusy AND NOT fbRequestSwitch1.bBusy AND NOT fbRequestSwitch2.bBusy AND NOT fbRequestSwitch3.bBusy THEN
		bError:= TRUE;
		
		IF NOT fbRequestSwitch0.bError THEN				 
			bGetContentResult:= fbRequestSwitch0.GetContent(pContent:= ADR(sContentS0), nContentSize:= SIZEOF(sContentS0), bSetNullTermination:= TRUE);
			IF fbRequestSwitch0.nStatusCode >= 200 AND fbRequestSwitch0.nStatusCode < 300 THEN
				bGetJsonResult:= FALSE;
				jsonDoc:= fbRequestSwitch0.GetJsonDomContent(fbJson);
				IF jsonDoc <> 0 THEN
					bGetJsonResult:= TRUE;
					IF fbJson.HasMember(jsonDoc, 'output')  THEN
						jsonVal:= fbJson.FindMember(jsonDoc, 'apower');
						nValidResCount:= nValidResCount+1;
						IF fbJson.IsDouble(jsonVal) THEN							
							lrapowerP1:= fbJson.GetDouble(jsonVal);									
						END_IF
						jsonVal:= fbJson.FindMember(jsonDoc, 'voltage');
						nValidResCount:= nValidResCount+1;					
						IF fbJson.IsDouble(jsonVal) THEN							
							lrvoltageP1:= fbJson.GetDouble(jsonVal);									
						END_IF
						jsonVal:= fbJson.FindMember(jsonDoc, 'aenergy');
                        IF fbJson.HasMember(jsonVal, 'total') THEN
                            jsonVal:= fbJson.FindMember(jsonVal, 'total');
                            nValidResCount:= nValidResCount+1;
                            IF fbJson.IsDouble(jsonVal) THEN
                                lraenergyP1:= fbJson.GetDouble(jsonVal);
                            END_IF
						bError:= FALSE;
						END_IF
					END_IF						
				nResCount:= nResCount+1;			
				END_IF
			END_IF
		END_IF
		
		IF NOT fbRequestSwitch1.bError THEN				 
			bGetContentResult:= fbRequestSwitch1.GetContent(pContent:= ADR(sContentS1), nContentSize:= SIZEOF(sContentS1), bSetNullTermination:= TRUE);
			IF fbRequestSwitch1.nStatusCode >= 200 AND fbRequestSwitch1.nStatusCode < 300 THEN
				bGetJsonResult:= FALSE;
				jsonDoc:= fbRequestSwitch1.GetJsonDomContent(fbJson);
				IF jsonDoc <> 0 THEN
					bGetJsonResult:= TRUE;
					IF fbJson.HasMember(jsonDoc, 'output')  THEN
						jsonVal:= fbJson.FindMember(jsonDoc, 'apower');
						nValidResCount:= nValidResCount+1;
						IF fbJson.IsDouble(jsonVal) THEN							
							lrapowerP2:= fbJson.GetDouble(jsonVal);									
						END_IF
						jsonVal:= fbJson.FindMember(jsonDoc, 'voltage');
						nValidResCount:= nValidResCount+1;					
						IF fbJson.IsDouble(jsonVal) THEN							
							lrvoltageP2:= fbJson.GetDouble(jsonVal);									
						END_IF
						jsonVal:= fbJson.FindMember(jsonDoc, 'aenergy');
                        IF fbJson.HasMember(jsonVal, 'total') THEN
                            jsonVal:= fbJson.FindMember(jsonVal, 'total');
                            nValidResCount:= nValidResCount+1;
                            IF fbJson.IsDouble(jsonVal) THEN
                                lraenergyP2:= fbJson.GetDouble(jsonVal);
                            END_IF
						bError:= FALSE;
						END_IF
					END_IF						
				nResCount:= nResCount+1;			
				END_IF
			END_IF
		END_IF
		
		IF NOT fbRequestSwitch2.bError THEN				 
			bGetContentResult:= fbRequestSwitch2.GetContent(pContent:= ADR(sContentS2), nContentSize:= SIZEOF(sContentS2), bSetNullTermination:= TRUE);
			IF fbRequestSwitch2.nStatusCode >= 200 AND fbRequestSwitch2.nStatusCode < 300 THEN
				bGetJsonResult:= FALSE;
				jsonDoc:= fbRequestSwitch2.GetJsonDomContent(fbJson);
				IF jsonDoc <> 0 THEN
					bGetJsonResult:= TRUE;
					IF fbJson.HasMember(jsonDoc, 'output')  THEN
						jsonVal:= fbJson.FindMember(jsonDoc, 'apower');
						nValidResCount:= nValidResCount+1;
						IF fbJson.IsDouble(jsonVal) THEN							
							lrapowerP3:= fbJson.GetDouble(jsonVal);									
						END_IF
						jsonVal:= fbJson.FindMember(jsonDoc, 'voltage');
						nValidResCount:= nValidResCount+1;					
						IF fbJson.IsDouble(jsonVal) THEN							
							lrvoltageP3:= fbJson.GetDouble(jsonVal);									
						END_IF
						jsonVal:= fbJson.FindMember(jsonDoc, 'aenergy');
                        IF fbJson.HasMember(jsonVal, 'total') THEN
                            jsonVal:= fbJson.FindMember(jsonVal, 'total');
                            nValidResCount:= nValidResCount+1;
                            IF fbJson.IsDouble(jsonVal) THEN
                                lraenergyP3:= fbJson.GetDouble(jsonVal);
                            END_IF
						bError:= FALSE;
						END_IF
					END_IF						
				nResCount:= nResCount+1;			
				END_IF
			END_IF
		END_IF
		
		IF NOT fbRequestSwitch3.bError THEN				 
			bGetContentResult:= fbRequestSwitch3.GetContent(pContent:= ADR(sContentS3), nContentSize:= SIZEOF(sContentS3), bSetNullTermination:= TRUE);
			IF fbRequestSwitch3.nStatusCode >= 200 AND fbRequestSwitch3.nStatusCode < 300 THEN
				bGetJsonResult:= FALSE;
				jsonDoc:= fbRequestSwitch3.GetJsonDomContent(fbJson);
				IF jsonDoc <> 0 THEN
					bGetJsonResult:= TRUE;
					IF fbJson.HasMember(jsonDoc, 'output')  THEN
						jsonVal:= fbJson.FindMember(jsonDoc, 'apower');
						nValidResCount:= nValidResCount+1;
						IF fbJson.IsDouble(jsonVal) THEN							
							lrapowerP4:= fbJson.GetDouble(jsonVal);									
						END_IF
						jsonVal:= fbJson.FindMember(jsonDoc, 'voltage');
						nValidResCount:= nValidResCount+1;					
						IF fbJson.IsDouble(jsonVal) THEN							
							lrvoltageP4:= fbJson.GetDouble(jsonVal);									
						END_IF
						jsonVal:= fbJson.FindMember(jsonDoc, 'aenergy');
                        IF fbJson.HasMember(jsonVal, 'total') THEN
                            jsonVal:= fbJson.FindMember(jsonVal, 'total');
                            nValidResCount:= nValidResCount+1;
                            IF fbJson.IsDouble(jsonVal) THEN
                                lraenergyP4:= fbJson.GetDouble(jsonVal);
                            END_IF
						bError:= FALSE;
						END_IF
					END_IF						
				nResCount:= nResCount+1;			
				END_IF
			END_IF
		END_IF
		
	nState:= 0;
	bBusy:= FALSE;
		IF bError THEN
			nErrCount:= nErrCount+1;
		END_IF
	END_IF  	
END_CASE

fbClient.Execute();

END_FUNCTION_BLOCK

// ---- POUs/Logic.TcPOU
PROGRAM Logic
VAR
	FB_MBUS_EMH_DIZ_0: FB_MBUS_EMH_DIZ;
	FB_MBUSKL6781_0: FB_MBUSKL6781;
	mStart: BOOL;
	stComIn  AT%I*: ST_KL6781inData22B;
	stComOut AT%Q*: ST_KL6781outData22B;
	stCom    : ST_MBUS_Communication;
	mDisabled: BOOL;
	R_TRIG_0: r_trig;
	string_Error: E_MBUS_Error;
	string_Error_OK: E_MBUS_Error;
	mTriggered: BOOL;
END_VAR

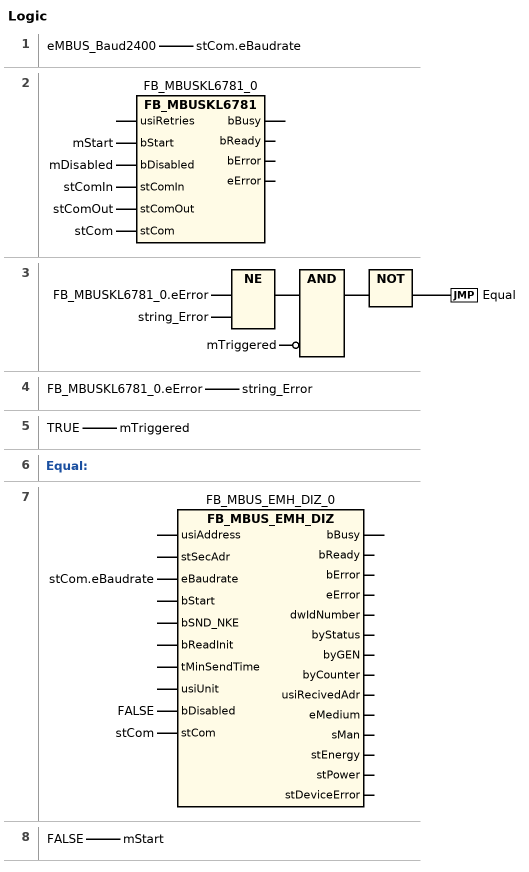
// NETWORK 1
stCom.eBaudrate := eMBUS_Baud2400;

// NETWORK 2
FB_MBUSKL6781_0(
    bStart := mStart,
    bDisabled := mDisabled,
    stComIn := stComIn,
    stComOut := stComOut,
    stCom := stCom); // FB_MBUSKL6781

// NETWORK 3
IF NOT (FB_MBUSKL6781_0.eError <> string_Error AND NOT mTriggered) THEN JMP Equal; END_IF

// NETWORK 4
string_Error := FB_MBUSKL6781_0.eError;

// NETWORK 5
mTriggered := TRUE;

// NETWORK 6
Equal: ;

// NETWORK 7
FB_MBUS_EMH_DIZ_0(eBaudrate := stCom.eBaudrate, bDisabled := FALSE, stCom := stCom); // FB_MBUS_EMH_DIZ

// NETWORK 8
mStart := FALSE;

END_PROGRAM

// ---- POUs/prgSmartMeter.TcPOU
PROGRAM prgSmartMeter
VAR
//	fbSmartMeter	: FB_KL6781_MBus_Master;	
	int_LiveCount		: INT;	//{#lynus.ag#()}
END_VAR

// fbSmartMeter(eBaudrateMBus := 9600);
logic ();
int_LiveCount:=int_LiveCount+1;

END_PROGRAM
